// TwinCAT 3 PLC project PlC
// ProgramVersion: 3.1.4023.0
// libraries:
//   EfficientIO Communicator, * (EfficientIO)
//   Tc2_Standard, * (Beckhoff Automation GmbH)
//   Tc2_System, * (Beckhoff Automation GmbH)
//   Tc3_Module, * (Beckhoff Automation GmbH)
// project tree:
//   GVLs/ GVL.TcGVL
//   / PlcTask.TcTTO, PlcTaskFast.TcTTO
//   VISUs/POUs/ prgComEffIO.TcPOU, prgMain.TcPOU, prgRWEffIO.TcPOU, prgVarEffIO.TcPOU
// real-time tasks:
//   TASK PlcTask: cycle T#10ms, priority 20, ADS port 350
//   TASK PlcTaskFast: cycle T#5ms, priority 21, ADS port 351

CONFIGURATION PlC
    RESOURCE PLC ON TwinCAT3
        TASK PlcTask(INTERVAL := T#10ms, PRIORITY := 20);
        TASK PlcTaskFast(INTERVAL := T#5ms, PRIORITY := 21);
        PROGRAM prgMain WITH PlcTask : prgMain;
        PROGRAM prgComEffIO WITH PlcTask : prgComEffIO;
        PROGRAM prgRWEffIO WITH PlcTaskFast : prgRWEffIO;
        PROGRAM prgVarEffIO WITH PlcTaskFast : prgVarEffIO;
    END_RESOURCE
END_CONFIGURATION

// ---- GVLs/GVL.TcGVL
{attribute 'qualified_only'}
VAR_GLOBAL
	mb_Input_Registers   :ARRAY[0..20] OF INT;	// Modbus Adress 32768 Funciton Code 04
END_VAR

// ---- VISUs/POUs/prgMain.TcPOU
PROGRAM prgMain
VAR
//	intLiveCount			: INT;				//{#lynus.ag#()}
	intArray  AT%MB0        :ARRAY[0..255] OF INT;		//Modbus Adress list for GLT (writing from GLT to Efficient IO)
														// --> output from Efficient IO to GLT in GVL.mb_Input_Registers
	
	TON_HeartBeat1: TON;
	TON_HeartBeat2: TON;
	real_RoomTemperature_409: REAL;			//{#lynus.ag#()}
	real_RoomTemperature_210: REAL;			//{#lynus.ag#()}
	bool_Mode_Zone_East_Off: BOOL;			//{#lynus.ag#()}
	bool_Mode_Zone_East_Cooling: BOOL;		//{#lynus.ag#()}
	bool_Mode_Zone_East_Heating: BOOL;		//{#lynus.ag#()}
	int_Mode_Zone_East: INT;				//{#lynus.ag#()}
	real_SupplyTempEast: REAL;				//{#lynus.ag#()}
	real_RoomTemperature_404: REAL;			//{#lynus.ag#()}
	real_RoomTemperature_204: REAL;			//{#lynus.ag#()}
	bool_Mode_Zone_West_Off: BOOL;			//{#lynus.ag#()}
	bool_Mode_Zone_West_Cooling: BOOL;		//{#lynus.ag#()}
	bool_Mode_Zone_West_Heating: BOOL;		//{#lynus.ag#()}
	int_Mode_Zone_West: INT;				//{#lynus.ag#()}
	real_SupplyTempWest: REAL;				//{#lynus.ag#()}
	real_RoomTemperature_Meeting6OG: REAL;	//{#lynus.ag#()}
	real_RoomTemperature_DinningRoomSmall: REAL;	//{#lynus.ag#()}
	real_RoomTemperature_DinningRoom: REAL;	//{#lynus.ag#()}
	bool_Mode_Zone_West2_Off: BOOL;			//{#lynus.ag#()}
	bool_Mode_Zone_West2_Cooling: BOOL;		//{#lynus.ag#()}
	bool_Mode_Zone_West2_Heating: BOOL;		//{#lynus.ag#()}
	int_Mode_Zone_West2: INT;				//{#lynus.ag#()}
	real_SupplyTempWest2: REAL;				//{#lynus.ag#()}
	bool_SPHeartBeat: BOOL;					//{#lynus.ag#()}
	byte_SPErrorWarning:BYTE;				//{#lynus.ag#()}
	bool_SPREady: BOOL;						//{#lynus.ag#()}
	r_trig1: R_trig;
	f_trig1: f_trig;
	ton_HB_Check: Ton;
	
	real_AverageRoomTemp: REAL;				//{#lynus.ag#()}
END_VAR
VAR PERSISTENT
	bool_EnableHeartbeat		:BOOL;		//{#lynus.ag#()}
	bool_Enable_ZoneWest		:BOOL;		//{#lynus.ag#()}
	bool_Enable_ZoneEast		:BOOL;		//{#lynus.ag#()}
	bool_Enable_ZoneWest2		:BOOL;		//{#lynus.ag#()}
	real_Setpoint_ZoneWest		:REAL;		//{#lynus.ag#()}
	real_Setpoint_ZoneEast		:REAL;		//{#lynus.ag#()}
	real_Setpoint2_ZoneWest		:REAL;		//{#lynus.ag#()}
END_VAR

//Creator : Stefan Lackner
//Company : Efficient IO
//Date : 12.10.2022
//Version : 0.0.1.1

// Heartbeat Bit 0 changing every 30s
// MB Adress 12288 where the GLT writes into, MB Adress 32768 where the GLT reads with function code 4
// The Heartbeat will only get sent to the GLT, when the received enable bit is high and the 1m received HB from the SetPoint Optimizer is good


//The SP HeartBeat get checked for the rising and falling edge, if no change within 5m then the Heartbeat to the GLT gets canceled					
r_trig1(CLK:=bool_SPHeartBeat);
f_trig1(CLK:=bool_SPHeartBeat);

ton_HB_Check(	In:=NOT (r_trig1.Q OR f_trig1.Q),
				PT:=T#5M);							// timer gets reset with every falling/rising edge of the HB bit from the Setpointoptimizer
				
IF bool_EnableHeartbeat AND NOT ton_HB_Check.q THEN
	IF TON_HeartBeat1.Q THEN
		intArray[0]:=1;		// not used, see GVL.mb_Input_Registers
		GVL.mb_Input_Registers[0]:=1;
	ELSE
		intArray[0]:=0;		// not used, see GVL.mb_Input_Registers
		GVL.mb_Input_Registers[0]:=0;
	END_IF
END_IF
TON_HeartBeat1(	IN:= TRUE AND NOT TON_HeartBeat2.Q ,
		PT:= T#30S,
		Q=> );
TON_HeartBeat2(	IN:= TON_HeartBeat1.Q,
		PT:= T#30S);
		
// MB Adress 12298
real_RoomTemperature_409 	:= INT_TO_REAL (intArray[10])/10;
// MB Adress 12299
real_RoomTemperature_210 	:= INT_TO_REAL (intArray[11])/10;
// MB Adress 12300
CASE intArray[12] OF
	0:	
		bool_Mode_Zone_East_Off		:=TRUE;
		bool_Mode_Zone_East_Cooling	:=FALSE;
		bool_Mode_Zone_East_Heating	:=FALSE;
	1:	
		bool_Mode_Zone_East_Off		:=FALSE;
		bool_Mode_Zone_East_Cooling	:=TRUE;
		bool_Mode_Zone_East_Heating	:=FALSE;
	2:	
		bool_Mode_Zone_East_Off		:=FALSE;
		bool_Mode_Zone_East_Cooling	:=FALSE;
		bool_Mode_Zone_East_Heating	:=TRUE;
END_CASE
int_Mode_Zone_East	:=intArray[12];
// MB Adress 12301
real_SupplyTempEast			:= INT_TO_REAL (intArray[13])/10;
// MB Adress 12302
real_RoomTemperature_404 	:= INT_TO_REAL (intArray[14])/10;
// MB Adress 12303
real_RoomTemperature_204 	:= INT_TO_REAL (intArray[15])/10;
// MB Adress 12304
CASE intArray[16] OF
	0:	
		bool_Mode_Zone_West_Off		:=TRUE;
		bool_Mode_Zone_West_Cooling	:=FALSE;
		bool_Mode_Zone_West_Heating	:=FALSE;
	1:	
		bool_Mode_Zone_West_Off		:=FALSE;
		bool_Mode_Zone_West_Cooling	:=TRUE;
		bool_Mode_Zone_West_Heating	:=FALSE;
	2:	
		bool_Mode_Zone_West_Off		:=FALSE;
		bool_Mode_Zone_West_Cooling	:=FALSE;
		bool_Mode_Zone_West_Heating	:=TRUE;
END_CASE
int_Mode_Zone_West	:=intArray[16];
// MB Adress 12305
real_SupplyTempWest						:= INT_TO_REAL (intArray[17])/10;	
// MB Adress 12306
real_RoomTemperature_Meeting6OG 		:= INT_TO_REAL (intArray[18])/10;
// MB Adress 12307
real_RoomTemperature_DinningRoomSmall	:= INT_TO_REAL (intArray[19])/10;
// MB Adress 12308
real_RoomTemperature_DinningRoom		:= INT_TO_REAL (intArray[20])/10;
// MB Adress 12309
CASE intArray[21] OF
	0:	
		bool_Mode_Zone_West2_Off		:=TRUE;
		bool_Mode_Zone_West2_Cooling	:=FALSE;
		bool_Mode_Zone_West2_Heating	:=FALSE;
	1:	
		bool_Mode_Zone_West2_Off		:=FALSE;
		bool_Mode_Zone_West2_Cooling	:=TRUE;
		bool_Mode_Zone_West2_Heating	:=FALSE;
	2:	
		bool_Mode_Zone_West2_Off		:=FALSE;
		bool_Mode_Zone_West2_Cooling	:=FALSE;
		bool_Mode_Zone_West2_Heating	:=TRUE;
END_CASE
int_Mode_Zone_West2	:=intArray[21];
// MB Adress 12310
real_SupplyTempWest2 	:= INT_TO_REAL (intArray[22])/10;		


// received setpoints from AI
// MB Adress 12488-12490

intArray[200] := REAL_TO_INT(real_Setpoint_ZoneEast*10); 	// not used, see GVL.mb_Input_Registers
intArray[201] := REAL_TO_INT(real_Setpoint_ZoneWest*10); 	// not used, see GVL.mb_Input_Registers
intArray[202] := REAL_TO_INT(real_Setpoint2_ZoneWest*10); 	// not used, see GVL.mb_Input_Registers

gvl.mb_Input_Registers[1]:=intArray[200];
gvl.mb_Input_Registers[2]:=intArray[201];
gvl.mb_Input_Registers[3]:=intArray[202];


real_AverageRoomTemp := (real_RoomTemperature_409 + real_RoomTemperature_210 + real_RoomTemperature_404 + real_RoomTemperature_204 + real_RoomTemperature_Meeting6OG + real_RoomTemperature_DinningRoomSmall + real_RoomTemperature_DinningRoom) / 7;

// enable bit for each zone
IF bool_Enable_ZoneWest AND NOT ton_HB_Check.q THEN
	IF TON_HeartBeat1.Q THEN
		GVL.mb_Input_Registers[4]:=1;
	ELSE
		GVL.mb_Input_Registers[4]:=0;
	END_IF
END_IF
IF bool_Enable_ZoneEast AND NOT ton_HB_Check.q THEN
	IF TON_HeartBeat1.Q THEN
		GVL.mb_Input_Registers[5]:=1;
	ELSE
		GVL.mb_Input_Registers[5]:=0;
	END_IF
END_IF
IF bool_Enable_ZoneWest2 AND NOT ton_HB_Check.q THEN
	IF TON_HeartBeat1.Q THEN
		GVL.mb_Input_Registers[6]:=1;
	ELSE
		GVL.mb_Input_Registers[6]:=0;
	END_IF
END_IF

END_PROGRAM

// ---- VISUs/POUs/prgComEffIO.TcPOU
PROGRAM prgComEffIO
VAR
	fbCom		: FB_MqttCommunicator_V2;
END_VAR

fbCom(
	bConnect:= TRUE, 
	strAuthKey:= 'BE736352867778' , 
	sUserName:= '357937e6-a18b-481e-8d82-4d957ba896c8', 
	sUserPassword:= 'eb079f87-6065-4dfe-8b33-960e910d1962' , 
	eSavePositionCertificate:= eSavePositionOnPLC.ePostionHardDisk , 
	time_HeartBeat_sec:= , 
	bConnected=> , 
	bError=> , 
	hrErrorCode=> , 
	eConnectionState=> , 
	eErrorMessage_Out=> );

(* old
fbCom(
	bConnect:= TRUE, 
	sUserName:= '4bd5671c-5161-4477-be33-80f6ab0ab0ea', 
	sUserPassword:= 'a9f16306-5d85-4294-8f17-fbe4adf6f24f', 
	eSavePositionCertificate:= eSavePositionOnPLC.ePostionHardDisk, 
	bConnected=> , 
	bError=> , 
	hrErrorCode=> , 
	eConnectionState=> , 
	eErrorMessage_Out=> );
*)

END_PROGRAM

// ---- VISUs/POUs/prgRWEffIO.TcPOU
PROGRAM prgRWEffIO
VAR
	fbRW1		: FB_ReadWrite_V2;
END_VAR

fbRW1(
	eUploadType:= eSelectDataUploadType.e_Change_Intervall5min, 
	bBusy=> , 
	bError=> , 
	udiErrorCodeOut=> ,
	eErrorReadWrite_Out=> );

END_PROGRAM

// ---- VISUs/POUs/prgVarEffIO.TcPOU
PROGRAM prgVarEffIO
VAR
	fbVar		: FB_VarInfo;
END_VAR

fbVar(
	bReadInfo:= , 
	eTMCFile:= eSelectTMCFile.eDontUseTMCFile, 
	eSavePositionTMCFile:= eSavePositionOnPLC.ePostionHardDisk, 
	udiCounterFoundVariables=> , 
	bError=> , 
	bBusy=> , 
	byProgress=> , 
	udiErrorCodeOut=> , 
	eErrorVarInfo_Out=> , 
	sVarWithError=> );

END_PROGRAM
